(* Schneider Machine Expert - Basic project Scada_tram_1, file version 2.7.0.0 *)
(* ProjectInformations: Name=New project *)

HARDWARE
  Cpu 0: TM221CE24R
  EthernetConfiguration: NetworkName=M221, IpAllocationMode=FixedAddress, IpAddress=192.168.1.15, SubnetMask=255.255.255.0
  SerialLineConfiguration: Baud=Baud19200, Parity=ParityEven, DataBits=DataBits8, StopBits=StopBits1, PhysicalMedium=PhysicalMediumRs485, TransmissionMode=TransmissionModeModbusRtu, SlaveId=1, Addressing=SlaveAddressing
  MastTask: UsePeriodScanMode=false, PeriodScan=100
  FastTask: Period=255
  CpuBehavior: StartingMode=StartAsPreviousState, AutoSaveRamOnEeprom=true, WatchdogPeriod=250

SYMBOLS  (address, symbol, comment, settings)
  %M1       LOW_WATER
  %M2       AUTO_REMOTE
  %M3       LOCAL
  %M4       PROTECTED_PHASE
  %M5       RUN_SOFT_STATER_1
  %M6       RUN_SOFT_STATER_2
  %M7       ERROR_PUMB_1
  %M8       ERROR_PUMB_2
  %M11      RUN_PUMB_1
  %M12      RUN_PUMB_2
  %I0.1       "Low Water"
  %I0.2       "Auto/remote"
  %I0.3       "Local"
  %I0.4       "Protected phase"
  %I0.5       "Run soft stater 1"
  %I0.6       "Run soft stater 2"
  %I0.7       "Error pumb 1"
  %I0.8       "Error pumb 2"
  %Q0.1     COIL_RUN_PUMB_1
  %Q0.2     COIL_RUN_PUMB_2

POU Control tram 1
  (* SectionNumber=1 *)

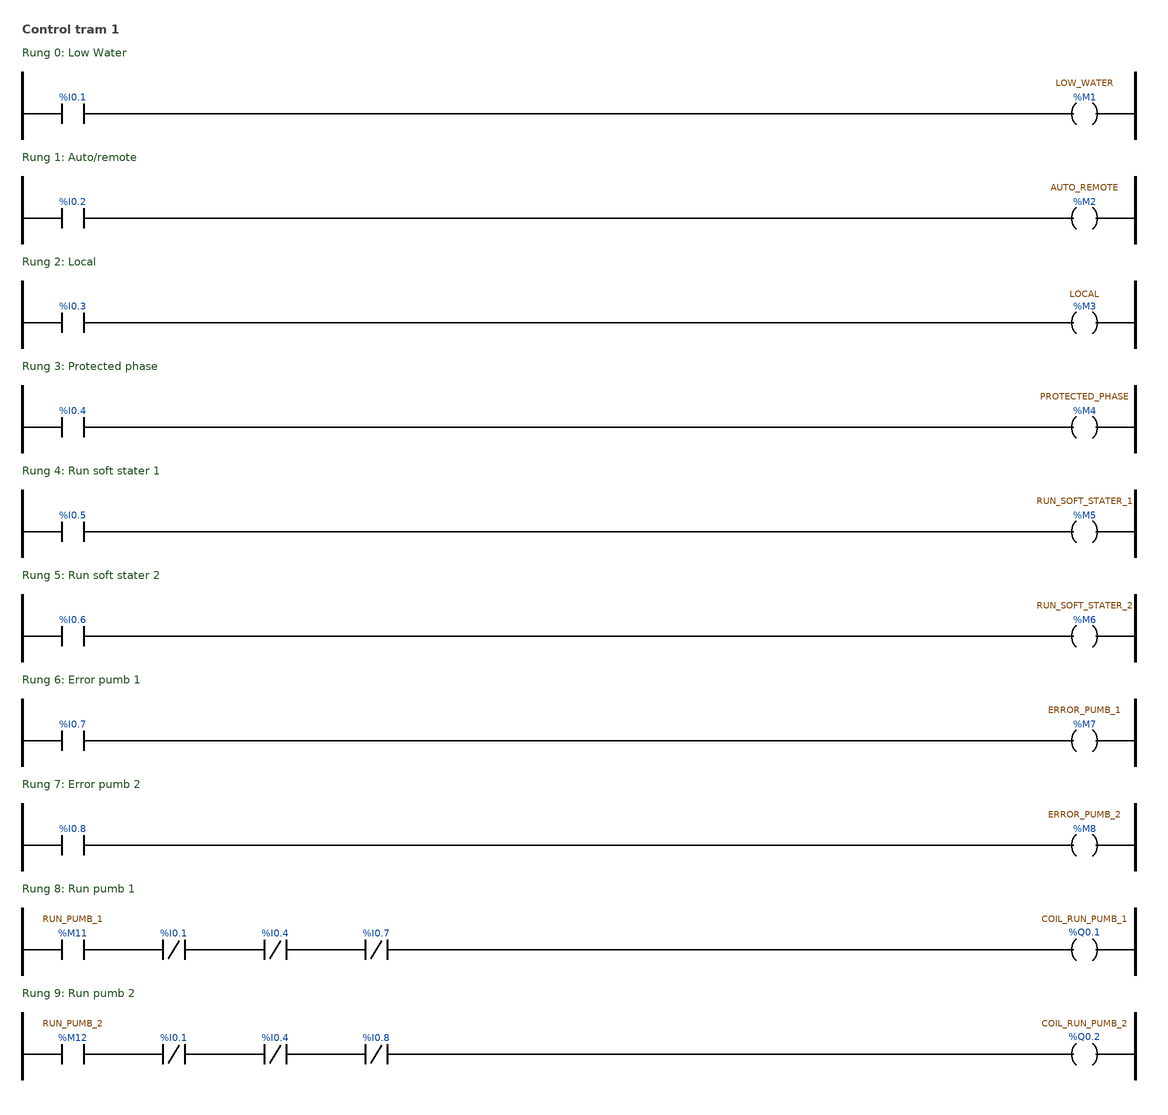

// Rung 0: Low Water
  LD %I0.1
  ST %M1                  (* LOW_WATER *)
  // as ST:
  //   LOW_WATER := %I0.1;

// Rung 1: Auto/remote
  LD %I0.2
  ST %M2                  (* AUTO_REMOTE *)
  // as ST:
  //   AUTO_REMOTE := %I0.2;

// Rung 2: Local
  LD %I0.3
  ST %M3                  (* LOCAL *)
  // as ST:
  //   LOCAL := %I0.3;

// Rung 3: Protected phase
  LD %I0.4
  ST %M4                  (* PROTECTED_PHASE *)
  // as ST:
  //   PROTECTED_PHASE := %I0.4;

// Rung 4: Run soft stater 1
  LD %I0.5
  ST %M5                  (* RUN_SOFT_STATER_1 *)
  // as ST:
  //   RUN_SOFT_STATER_1 := %I0.5;

// Rung 5: Run soft stater 2
  LD %I0.6
  ST %M6                  (* RUN_SOFT_STATER_2 *)
  // as ST:
  //   RUN_SOFT_STATER_2 := %I0.6;

// Rung 6: Error pumb 1
  LD %I0.7
  ST %M7                  (* ERROR_PUMB_1 *)
  // as ST:
  //   ERROR_PUMB_1 := %I0.7;

// Rung 7: Error pumb 2
  LD %I0.8
  ST %M8                  (* ERROR_PUMB_2 *)
  // as ST:
  //   ERROR_PUMB_2 := %I0.8;

// Rung 8: Run pumb 1
  LD %M11                 (* RUN_PUMB_1 *)
  ANDN %I0.1
  ANDN %I0.4
  ANDN %I0.7
  ST %Q0.1                (* COIL_RUN_PUMB_1 *)
  // as ST:
  //   COIL_RUN_PUMB_1 := RUN_PUMB_1 AND NOT %I0.1 AND NOT %I0.4 AND NOT %I0.7;

// Rung 9: Run pumb 2
  LD %M12                 (* RUN_PUMB_2 *)
  ANDN %I0.1
  ANDN %I0.4
  ANDN %I0.8
  ST %Q0.2                (* COIL_RUN_PUMB_2 *)
  // as ST:
  //   COIL_RUN_PUMB_2 := RUN_PUMB_2 AND NOT %I0.1 AND NOT %I0.4 AND NOT %I0.8;
